INTERFACE IAxisIAI

PROPERTY DriveRef : REFERENCE TO AxisIAI
GET
END_GET
END_PROPERTY

END_INTERFACE

(* stored: Version 1.1.0.1, ProductVersion 3.1.4024.12
   Itf IAxisIAI: Id {afe947c1-2a9f-4545-83f8-6a383e4eba28}
   Property DriveRef: Id {0f1bd579-7aa1-47ee-bc4d-f5e57bd343eb}
   Get Get: Id {e762046f-ecd7-4480-89be-748032735750} *)
